{attribute 'GeneratedUsingTerminal: EL6201-0000-0017'}
{attribute addProperty BoxType "EL6201-0000-0017"}
{attribute addProperty Id "Slave_20A_DI0BOOL1Slave_20A_DI1BOOL1Slave_20A_DI2BOOL1Slave_20A_DI3BOOL1Slave_20B_DI0BOOL1Slave_20B_DI1BOOL1Slave_20B_DI2BOOL1Slave_20B_DI3BOOL1"}
{attribute addProperty CRC "2546059930"}
{attribute addProperty Size "8"}
TYPE Slave_20_Inputs_97C1CA9A :
STRUCT
	{attribute addProperty Name "Slave_20A_DI0"}
	Slave_20A_DI0 : BOOL;
	{attribute addProperty Name "Slave_20A_DI1"}
	Slave_20A_DI1 : BOOL;
	{attribute addProperty Name "Slave_20A_DI2"}
	Slave_20A_DI2 : BOOL;
	{attribute addProperty Name "Slave_20A_DI3"}
	Slave_20A_DI3 : BOOL;
	{attribute addProperty Name "Slave_20B_DI0"}
	Slave_20B_DI0 : BOOL;
	{attribute addProperty Name "Slave_20B_DI1"}
	Slave_20B_DI1 : BOOL;
	{attribute addProperty Name "Slave_20B_DI2"}
	Slave_20B_DI2 : BOOL;
	{attribute addProperty Name "Slave_20B_DI3"}
	Slave_20B_DI3 : BOOL;
END_STRUCT
END_TYPE

(* stored: Version 1.2.0.0, ProductVersion 3.1.4024.11
   DUT Slave_20_Inputs_97C1CA9A: Id {305c8601-4e5d-4f8e-a19b-c72f7ac64552} *)
